(* IEC 61131-3 sources: plc-browser-io/CODESYSv3/CODESYS_Control_Win_V3_x64/Application/Logger, 3 files *)

(* ---- LogComponent.st ---- *)
{attribute 'qualified_only'}
{attribute 'symbol' := 'none'}
VAR_GLOBAL
	RTM		   : STRING := 'Runtime'; //Runtime events
	WS		   : STRING := 'WebSocket'; //WebSocket server log

	Logger     : Logger;  //Instance of logger component
END_VAR

(* ---- Logger.st ---- *)
FUNCTION_BLOCK Logger
VAR_INPUT
END_VAR
VAR_OUTPUT
END_VAR
VAR
	message  : STRING;
	udiCmpId : UDINT;
	cmResult : Component_Manager.SysTypes.RTS_IEC_RESULT;
END_VAR

// === IMPLEMENTATION ===
//Register components
CMAddComponent2( pszComponent := LogComponent.RTM
               , udiVersion   := 16#01
               , udiCmpId     := ADR(udiCmpId)
               , pResult      := ADR(cmResult));

CMAddComponent2( pszComponent := LogComponent.WS
               , udiVersion   := 16#01
               , udiCmpId     := ADR(udiCmpId)
               , pResult      := ADR(cmResult));

(* ---- Logger.LogADD.st ---- *)
(*
Add new record in logfile
Component: STRING from Component. Example: Component:= Component.user_action
LogClass: cmplog.LogClass. Example: LogClass:=cmplog.LogClass.LOG_ERROR
Message: STRING. Write here your Log Message.
*)

// LOG-file path: /var/opt/codesys/codesyscontrol.log

METHOD LogADD : BOOL
VAR_INPUT
	Component : STRING;
	LogClass  : UDINT;
	Message   : STRING := 'something happened';
END_VAR

// === IMPLEMENTATION ===
Component_Manager.CMAddComponent2(Component, 16#01, ADR(udiCmpId), ADR(cmResult));

CmpLog.LogAdd2(cmplog.LogConstants.STD_LOGGER, udiCmpID, LogClass, cmpErrors.Errors.ERR_FAILED, 0, Message);
